{attribute 'qualified_only'}
{attribute 'strict'}
TYPE E_IO2_InputSource :
(
	SENSOR	:= 1,
	MACHINE := 2
);
END_TYPE

(* stored: Version 1.1.0.1
   DUT E_IO2_InputSource: Id {099b6949-6097-4cc5-b902-d4f02cce430f} *)
